// TwinCAT 3 PLC project MainProgram
// ProgramVersion: 3.1.4023.0
// libraries:
//   Tc2_Standard, * (Beckhoff Automation GmbH)
//   Tc2_System, * (Beckhoff Automation GmbH)
//   Tc3_Module, * (Beckhoff Automation GmbH)
// project tree:
//   GVLs/ GVL_IO.TcGVL
//   / PlcTask.TcTTO
//   POUs/Devices/Beckhoff/ EL1008.TcPOU
//   POUs/Devices/Generic/ TwoStateSwitch.TcPOU
//   POUs/IO/ DigitalInputChannel.TcPOU, AssignableDigitalInputChannel.TcPOU, NullDigitalInputChannel.TcPOU, I_DigitalInput.TcIO
//   POUs/ MAIN.TcPOU
// real-time tasks:
//   TASK PlcTask: cycle T#10ms, priority 20, ADS port 350

CONFIGURATION MainProgram
    RESOURCE PLC ON TwinCAT3
        TASK PlcTask(INTERVAL := T#10ms, PRIORITY := 20);
        PROGRAM MAIN WITH PlcTask : MAIN;
    END_RESOURCE
END_CONFIGURATION

// ---- GVLs/GVL_IO.TcGVL
VAR_GLOBAL
	

	nullInputChannel : NullDigitalInputChannel;
	
	device1 : EL1008;
	
	myFanControlDigitalInput : AssignableDigitalInputChannel(nullInputChannel);
	
	myFanControl : TwoStateSwitch(myFanControlDigitalInput);

END_VAR

// ---- POUs/IO/I_DigitalInput.TcIO
INTERFACE I_DigitalInput

PROPERTY PUBLIC State : BOOL
GET
END_GET
END_PROPERTY

END_INTERFACE

// ---- POUs/MAIN.TcPOU
PROGRAM MAIN
VAR
	myDebug : BOOL;
	ChangeTo1 : BOOL;
	ChangeTo2 : BOOL;
END_VAR

IF myFanControl.IsOn THEN
	myDebug := TRUE;
ELSE 
	myDebug := FALSE;
END_IF

IF ChangeTo1 THEN
	ChangeTo1 := FALSE;
	myFanControlDigitalInput.ChangeDigitalInput(device1.GetDigitalInput(0));
END_IF

IF ChangeTo2 THEN
	ChangeTo2 := FALSE;
	myFanControlDigitalInput.ChangeDigitalInput(device1.GetDigitalInput(1));
END_IF

END_PROGRAM

// ---- POUs/IO/NullDigitalInputChannel.TcPOU
FUNCTION_BLOCK NullDigitalInputChannel implements I_DigitalInput

PROPERTY PUBLIC State : BOOL
GET
State := FALSE;
END_GET
END_PROPERTY

END_FUNCTION_BLOCK

// ---- POUs/Devices/Beckhoff/EL1008.TcPOU
FUNCTION_BLOCK EL1008
VAR
	Channels : ARRAY [0..7] OF DigitalInputChannel;
END_VAR

METHOD PUBLIC GetDigitalInput : I_DigitalInput
VAR_INPUT
	channelNumber : INT;
END_VAR
GetDigitalInput := Channels[channelNumber];
END_METHOD

END_FUNCTION_BLOCK

// ---- POUs/IO/DigitalInputChannel.TcPOU
FUNCTION_BLOCK DigitalInputChannel IMPLEMENTS I_DigitalInput
VAR
	input AT %I* : BOOL;
END_VAR

PROPERTY PUBLIC State : BOOL
GET
State := input;
END_GET
END_PROPERTY

END_FUNCTION_BLOCK

// ---- POUs/IO/AssignableDigitalInputChannel.TcPOU
FUNCTION_BLOCK AssignableDigitalInputChannel implements I_DigitalInput
VAR
	digitalInput : I_DigitalInput;
END_VAR

METHOD PUBLIC ChangeDigitalInput
VAR_INPUT
	DigitalInput : I_DigitalInput;
END_VAR
IF DigitalInput <> 0 THEN
	THIS^.digitalInput := DigitalInput;
END_IF
END_METHOD

METHOD FB_init : BOOL
VAR_INPUT
	bInitRetains : BOOL; // if TRUE, the retain variables are initialized (warm start / cold start)
	bInCopyCode : BOOL;  // if TRUE, the instance afterwards gets moved into the copy code (online change)
	DigitalInput : I_DigitalInput;
END_VAR
this^.digitalInput := DigitalInput;
END_METHOD

PROPERTY PUBLIC State : BOOL
GET
State := digitalInput.State;
END_GET
END_PROPERTY

END_FUNCTION_BLOCK

// ---- POUs/Devices/Generic/TwoStateSwitch.TcPOU
FUNCTION_BLOCK TwoStateSwitch
VAR
	digitalInput : I_DigitalInput;
END_VAR

METHOD FB_init : BOOL
VAR_INPUT
	bInitRetains : BOOL; // if TRUE, the retain variables are initialized (warm start / cold start)
	bInCopyCode : BOOL;  // if TRUE, the instance afterwards gets moved into the copy code (online change)
	DigitalInput : I_DigitalInput;
END_VAR
this^.digitalInput := DigitalInput;
END_METHOD

PROPERTY PUBLIC IsOn : BOOL
GET
IsOn := digitalInput.State;
END_GET
END_PROPERTY

END_FUNCTION_BLOCK
